PROGRAM P_AllStateChecker
VAR
	(*
		Author - Gideon Jgordon (GJ)
		Changes 
		-(GJ) stGSM moved here
	*)	
	bAllOk : BOOL;	// All OK process
	//bSAT_OK: BOOL;  //SAT Process OK
END_VAR


IF P_GeneralStateManager.nStateGeneral =GeneralStateMain.State_ErrorCheck THEN
	gvl.stGSM.bStop			:=TRUE;
	gvl.stGSM.bOverride		:=FALSE;
	gvl.stGSM.bStart		:=FALSE;
	gvl.stGSM.bReset		:=TRUE;	
END_IF

IF P_GeneralStateManager.nStateGeneral =GeneralStateMain.State_Init THEN
	gvl.stGSM.bStop		   :=TRUE;
	gvl.stGSM.bOverride	   :=TRUE;
	gvl.stGSM.bStart	   :=FALSE;
	gvl.stGSM.bReset	   :=FALSE;	
END_IF

IF P_GeneralStateManager.nStateGeneral =GeneralStateMain.State_Reset THEN
	gvl.stGSM.bStop		   :=TRUE;
	gvl.stGSM.bOverride	   :=FALSE;
	gvl.stGSM.bStart	   :=FALSE;
	gvl.stGSM.bReset	   :=TRUE;	
END_IF

IF P_GeneralStateManager.nStateGeneral =GeneralStateMain.State_Run THEN
	gvl.stGSM.bStop		   :=TRUE;
	gvl.stGSM.bOverride	   :=FALSE;
	gvl.stGSM.bStart	   :=FALSE;
	gvl.stGSM.bReset	   :=FALSE;
END_IF

IF P_GeneralStateManager.nStateGeneral =GeneralStateMain.State_Stop THEN
	gvl.stGSM.bStop		   :=TRUE;
	gvl.stGSM.bOverride	   :=FALSE;
	gvl.stGSM.bStart	   :=FALSE;
	gvl.stGSM.bReset	   :=FALSE;
END_IF

IF  	P_Feeder.bFeederOK 
	AND P_SheetAlignTable.bSAT_OK 
	AND P_VacummBeltTable.bVBT_OK
	AND P_EjectionGate.bEJ_OK
	AND P_StackerBeltTable.bSBT_OK		THEN
	bAllok:=TRUE;
ELSE
	bAllok:=FALSE;	
END_IF

END_PROGRAM

(* stored: Version 1.1.0.1, ProductVersion 3.1.4024.12
   POU P_AllStateChecker: Id {985017dc-d89e-49af-aaa8-dfefe2cd487c}, SpecialFunc None *)
